// TIA Portal V18 export
FUNCTION "BoilerModesCtrlAutoMode" : Void   // FC60106, LAD
{ S7_Optimized_Access := 'TRUE' }
VERSION : 0.1
// stored: AutoNumber false, IsIECCheckEnabled false, SetENOAutomatically false, UDAEnableTagReadback false
   VAR_INPUT
      cPreselectedPLCOpMode : Byte;
      cSchedulerTargetOpMode : Byte;
      cPanelSelectorActualMode : Byte;
   END_VAR
   VAR_OUTPUT
      cTargetOpMode : Byte;
      cActualOpMode : Byte;
   END_VAR
   VAR_TEMP
      TargetUnitMode_old : Int;
      ResetActualOperationMode : Bool;
   END_VAR
BEGIN

REGION Network 1 (SCL)
   CASE #cPanelSelectorActualMode OF
       0:                                                     // Switch is in Summer/OFF
           #cTargetOpMode := 0;                               //Summer
       1:                                                     // ON
           #cTargetOpMode := 1;                               // Winter 
       ELSE                                                   // Switch is in Auto
           IF #cPreselectedPLCOpMode = 2 THEN                 // PLC mode 2=Scheduler
               #cTargetOpMode := #cSchedulerTargetOpMode;     // 
           ELSE                                               //mode-0-1-2-
               #cTargetOpMode := #cPreselectedPLCOpMode;
           END_IF;
   END_CASE;
END_REGION

REGION Network 2 (SCL)
   IF #cTargetOpMode <> #cActualOpMode THEN
       // Update Actual OP Mode
       #cActualOpMode := #cTargetOpMode;
   END_IF;
END_REGION

REGION Network 3 (SCL)
   IF #cActualOpMode <> "cActualOpModePrevOne" THEN
       "iActualOpModeCounter" := "iActualOpModeCounter" + 1;
   END_IF;
END_REGION
END_FUNCTION
